TYPE St_Assy_Base :
STRUCT
	sSfc		:STRING;
	iOpIndex	:INT;
END_STRUCT
END_TYPE

(* stored: Version 1.1.0.1
   DUT St_Assy_Base: Id {5c11eaa4-3dd1-4205-bc54-b4a7a73d114d} *)
